TYPE SystemParameters :
STRUCT
	Operation: SystemOperationParameters;
	Defrost: DefrostParameters;
	Exercise: ExerciseParameters;
	SystemTime: STRING;
	ProjectDefaultSet: BOOL;
	{attribute 'TcEncoding':='UTF-8'}
	Diagram: string[80];
END_STRUCT
END_TYPE

(* stored: Version 1.1.0.1, ProductVersion 3.1.4024.6
   DUT SystemParameters: Id {7f9a91cd-9a6a-4f99-a168-e71b2e0fadb0} *)
